Fanuc KAREL source: kb00015.KL

-- PROVISIONAL review KL for V940-1; original PC SHA256 908b0efbf64c220ddba623af9a351291acc9a5bf2f8ca5c341f7c0d2497e5b2f
-- Incomplete behavior may be omitted. Consult companion uncertainty JSON. Do not deploy.
PROGRAM KB00015
%NOLOCKGROUP
BEGIN
  -- V9_ZERO_TABLE_METADATA_HINT layout=0002_ascii; no indexed target words; source/name/runtime held
  -- UNRESOLVED_PC offsets 5-14; opcodes 3F,75
  -- UNRESOLVED_PC offsets 19-26; opcodes 9D,23
  -- UNRESOLVED_PC offsets 31-49; opcodes 27,22,2A,22,31
  -- UNRESOLVED_PC offsets 54-58; opcodes 7F
END KB00015
